# EPICS autosave request: iocBoot/ioc3/auto_settings.req
file dbSave/23i_BP_Kb_.req  DIR=dbSave
file dbSave/23i_BP_Mo_.req  DIR=dbSave
file dbSave/23i_CS_Ah_.req  DIR=dbSave
file dbSave/23i_CS_Av_.req  DIR=dbSave
file dbSave/23i_KB_Hy_.req  DIR=dbSave
file dbSave/23i_KB_Hz_.req  DIR=dbSave
file dbSave/23i_KB_Vy_.req  DIR=dbSave
file dbSave/23i_KB_Vz_.req  DIR=dbSave
file dbSave/23i_MO_En_.req  DIR=dbSave
file dbSave/23i_MO_Ps_.req  DIR=dbSave
file dbSave/23i_MO_Tn1_.req DIR=dbSave
file dbSave/23i_MO_Tn2_.req DIR=dbSave
file dbSave/23i_WS_Ah_.req  DIR=dbSave
file dbSave/23i_WS_Av_.req  DIR=dbSave
%
